Yaskawa INFORM job: BATMAN_2STR2.JBI

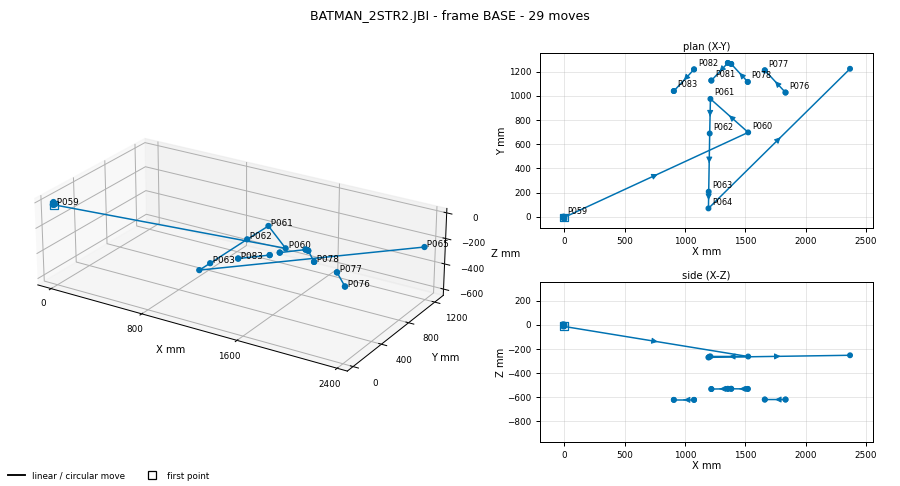
[picture p0: tool path of BATMAN_2STR2.JBI in frame BASE, 29 of 158 moves have a stored position in this frame; points joined in program order, loops and branches not executed]
/JOB
//NAME BATMAN_2STR2
///FOLDERNAME KRIS-SCIANA
//POS
///NPOS 87,87,0,38,0,0
///TOOL 0
///POSTYPE PULSE
///LIMIT ON
///PULSE
C00000=31537,-23080,-24186,7401,81948,158244
C00001=-4439,-79004,-57355,2552,77563,145804
C00002=-4909,-70479,-49283,2592,76991,145631
C00003=-4909,-70121,-48408,2595,76637,145623
C00004=-4003,-74801,-52630,2527,76803,145940
C00005=11747,-84119,-56660,1324,74120,151337
C00006=17222,-83520,-55007,884,73335,153227
C00007=17222,-83075,-54091,884,72998,153224
C00008=32420,-90805,-60082,-370,72663,158498
C00009=38310,-87672,-56905,-859,72363,160549
C00010=38411,-86269,-54218,-871,71436,160589
C00011=52965,-90491,-59465,-2036,72753,165631
C00012=61358,-83938,-55903,-2664,74169,168512
C00013=61358,-82452,-52843,-2677,73046,168534
C00014=75499,-77158,-53728,-3596,76905,173310
C00015=83067,-67878,-47888,-4094,78394,175877
C00016=83067,-67594,-47168,-4098,78099,175887
C00017=88580,-61652,-44685,-4402,79910,177718
C00018=88580,-61316,-43770,-4406,79520,177731
C00019=86164,-72702,-59256,-4234,83063,176784
C00020=57917,-53619,-44002,17021,94716,124656
C00021=59918,-45185,-32120,16966,91065,125425
C00022=59918,-44935,-31368,16961,90745,125381
C00023=57173,-65270,-44444,16695,89007,124177
C00024=59200,-80263,-49588,16922,84240,124236
C00025=59200,-79912,-48884,16927,83998,124202
C00026=59200,-86069,-61854,16879,88616,124838
C00027=77293,-89843,-63362,18058,83781,130525
C00028=78815,-87617,-60670,18129,82952,130941
C00029=78815,-87165,-59720,18140,82615,130890
C00030=77659,-102730,-69319,18171,80880,130220
C00031=85944,-117290,-70372,18932,72559,131861
C00032=85944,-116620,-69416,18956,72327,131824
C00033=85944,-124960,-81218,18696,75154,132276
C00034=151728,-153076,-87491,-11017,48359,191211
C00035=147386,-140874,-75268,-10077,46618,189610
C00036=147386,-140130,-74447,-10096,46496,189624
C00037=159688,-133609,-76919,-12343,52845,193892
C00038=159864,-112518,-69307,-11535,58898,193269
C00039=159864,-111881,-68341,-11567,58637,193296
C00040=178833,-115187,-73178,-14901,62898,200003
C00041=185982,-107062,-64617,-16080,63162,202660
C00042=185982,-103029,-58312,-16337,61422,202917
C00043=185982,-102236,-57075,-16389,61082,202968
C00044=187292,-93406,-58139,-15875,66332,202702
C00045=183818,-68327,-44618,-14942,70095,200919
C00046=183818,-67914,-43663,-14975,69731,200966
C00047=189068,-78650,-56857,-15464,73225,202429
C00048=240783,-65694,-51653,-5278,84394,164569
C00049=221621,-56342,-41396,-1214,76392,158122
C00050=221621,-56290,-41244,-1214,76326,158123
C00051=221621,-55882,-40078,-1216,75818,158128
C00052=209855,-65296,-47790,155,75648,154049
C00053=204224,-59057,-42452,814,75603,152098
C00054=204224,-58710,-41499,814,75195,152094
C00055=190935,-63343,-46423,2338,76108,147494
C00056=187139,-57536,-42749,2753,76951,146198
C00057=187139,-57216,-41822,2757,76545,146190
C00058=175859,-57355,-44220,3949,78417,142345
C00059=173058,-50767,-39052,4222,78764,141391
C00060=173058,-50451,-38053,4227,78312,141376
C00061=163443,-45354,-36848,5138,80747,138159
C00062=164371,-41258,-32523,5059,80134,138455
C00063=164371,-41027,-31730,5064,79765,138439
C00064=152450,-34091,-30773,6086,83554,134518
C00065=152482,-28025,-24496,6089,82810,134493
C00066=152482,-27812,-23636,6093,82393,134472
C00067=149914,-23676,-21598,6293,83456,133647
C00068=149914,-23406,-20465,6299,82902,133618
C00069=149914,-25053,-28729,6272,87116,133828
C00070=211398,-84605,-64904,-36,76260,154581
C00071=220860,-58623,-44430,-1132,77083,157849
C00072=149914,-25053,-28729,6272,87116,133828
C00073=120676,-124875,-96295,8199,80135,123403
C00074=-4439,-79004,-57355,2552,77563,145804
C00075=-4965,-72448,-51023,2596,77053,145613
C00076=88570,-66783,-53472,-4371,82677,177617
C00077=72474,-62045,-52325,1456,86059,123431
C00078=73182,-61072,-47349,1438,83485,123645
C00079=40588,-105091,-66546,14786,85577,117999
C00080=66697,-107157,-67194,17695,79826,126223
C00081=61032,-151860,-79989,18635,65463,124242
C00082=7538,-133985,-77466,26458,61671,147261
C00083=57429,-136223,-75586,15192,52650,153109
C00084=59881,-140929,-66526,16624,44527,152732
C00085=106253,-180552,-90268,3429,33706,171973
C00086=22771,-69913,-65485,-4348,88446,177417
///LIMIT OFF
BC00000=149550,282370,904111
BC00001=226428,281090,543192
BC00002=226428,281090,543192
BC00003=226428,281090,543192
BC00004=226427,281091,543189
BC00005=226427,281091,543189
BC00006=226427,281091,543189
BC00007=226427,281091,543189
BC00008=226427,281091,543189
BC00009=226427,281091,543189
BC00010=226427,281091,543189
BC00011=226427,281091,543189
BC00012=226427,281091,543189
BC00013=226427,281091,543189
BC00014=226427,281091,543189
BC00015=226427,281091,543189
BC00016=226427,281091,543189
BC00017=226427,281091,543189
BC00018=226427,281091,543189
BC00019=226427,281091,543187
BC00020=226427,281092,543184
BC00021=225242,280682,546364
BC00022=225242,280682,546364
BC00023=225242,280682,546364
BC00024=225242,280682,546364
BC00025=225242,280682,546364
BC00026=225242,280682,546364
BC00027=225242,280682,546364
BC00028=225242,280682,546364
BC00029=225242,280682,546364
BC00030=225242,280682,546364
BC00031=225242,280682,546364
BC00032=225242,280682,546364
BC00033=225242,280682,546364
BC00034=225242,280682,546364
BC00035=225242,280682,546364
BC00036=225242,280682,546364
BC00037=225242,280682,546364
BC00038=225242,280682,546364
BC00039=225242,280682,546364
BC00040=225242,280682,546364
BC00041=225242,280682,546364
BC00042=225242,280682,546364
BC00043=225242,280682,546364
BC00044=225242,280682,546364
BC00045=225242,280682,546364
BC00046=225242,280682,546364
BC00047=225242,280682,546364
BC00048=226427,281091,543187
BC00049=226427,319126,543187
BC00050=226427,319126,543187
BC00051=226427,319126,543187
BC00052=226427,319126,543184
BC00053=226427,319126,543184
BC00054=226427,319126,543184
BC00055=226427,319126,543184
BC00056=226427,319126,543184
BC00057=226427,319126,543184
BC00058=226427,319126,543184
BC00059=226427,319125,543182
BC00060=226427,319125,543182
BC00061=226427,319125,543182
BC00062=226427,319125,543182
BC00063=226427,319125,543182
BC00064=226427,319125,543182
BC00065=226427,319125,543182
BC00066=226427,319125,543182
BC00067=226427,319125,543182
BC00068=226427,319125,543182
BC00069=226427,319125,543182
BC00070=226427,319125,543182
BC00071=226427,319125,543182
BC00072=226427,319125,543182
BC00073=226427,319125,543182
BC00074=226428,281090,543192
BC00075=226428,281090,543192
BC00076=226428,281090,543192
BC00077=226428,281090,543192
BC00078=226428,281090,543192
BC00079=228873,257687,554679
BC00080=228873,257687,554679
BC00081=229563,251082,557921
BC00082=133596,251082,557921
BC00083=134171,249919,558492
BC00084=134171,249919,558492
BC00085=134170,249920,558489
BC00086=134714,456554,904710
///POSTYPE BASE
///RECTAN
///RCONF 0,0,0,0,0,0,0,0,0,0,0,0,0,0,0,0,0,0,0,0,0,0,0,0
P00059=-2.448,-6.714,-12.718,0.0000,0.0000,0.0000
P00060=1524.284,698.404,-261.973,-0.4635,36.8346,-1.2388
P00061=1211.499,975.999,-261.374,0.5148,35.2356,175.5099
P00062=1205.574,689.500,-262.704,0.5159,35.2461,175.5270
P00063=1197.217,207.358,-268.729,0.4863,35.2395,175.4586
P00064=1195.199,68.975,-269.171,0.5092,35.2366,175.4908
P00065=2367.684,1225.356,-251.745,0.6375,35.5356,-175.5535
P00070=2.449,-18.318,2.615,0.0000,0.0000,0.0000
P00071=-2.048,-0.034,-9.092,0.0000,0.0000,0.0000
P00072=-1.595,-0.049,-6.373,0.0000,0.0000,0.0000
P00073=-8.474,-10.331,-11.894,0.0000,0.0000,0.0000
P00074=1.731,-3.007,-10.460,0.0000,0.0000,0.0000
///RCONF 0,1,0,0,0,0,0,0,0,0,0,0,0,0,0,0,0,0,0,0,0,0,0,0
P00075=-9.634,0.014,4.922,0.0000,0.0000,0.0000
///RCONF 0,0,0,0,0,0,0,0,0,0,0,0,0,0,0,0,0,0,0,0,0,0,0,0
P00076=1833.500,1028.615,-618.215,10.0256,37.5190,56.2681
P00077=1661.766,1212.555,-618.325,10.0309,37.5577,56.2858
P00078=1520.740,1116.757,-530.271,10.0398,37.5578,56.2925
P00079=1383.754,1265.334,-529.217,10.0293,37.5461,56.2787
P00080=1355.833,1273.708,-529.583,10.0283,37.5305,126.4716
P00081=1219.184,1127.874,-531.327,10.0137,37.5345,126.4324
P00082=1075.995,1220.294,-620.895,10.0203,37.5289,126.4576
P00083=908.434,1040.970,-620.895,10.0141,37.5419,126.4584
P00087=-17.000,-22.000,-3.000,0.0000,0.0000,0.0000
P00088=-8.588,-0.108,-11.097,0.0000,0.0000,0.0000
P00089=5.931,-12.286,-8.772,0.0000,0.0000,0.0000
P00090=-14.057,13.261,-6.464,0.0000,0.0000,0.0000
P00091=1.048,0.648,3.624,0.0000,0.0000,0.0000
P00092=12.000,-9.000,-4.000,0.0000,0.0000,0.0000
P00093=-12.000,12.000,-3.000,0.0000,0.0000,0.0000
P00094=10.000,10.000,-3.000,0.0000,0.0000,0.0000
P00095=-11.943,-14.820,-6.815,0.0000,0.0000,0.0000
P00096=-4.844,-19.262,-10.890,0.0000,0.0000,0.0000
P00108=0.000,0.000,-3.000,0.0000,0.0000,0.0000
P00123=0.000,-50.000,0.000,0.0000,0.0000,0.0000
P00125=0.000,0.000,2.400,0.0000,0.0000,0.0000
P00126=-50.000,0.000,0.000,0.0000,0.0000,0.0000
P00127=50.000,0.000,0.000,0.0000,0.0000,0.0000
P00172=2.000,-12.000,-3.000,0.0000,0.0000,40.0000
P00173=-5.000,-9.000,-2.400,0.0000,0.0000,-15.0000
//INST
///DATE 2024/07/30 17:34
///COMM NOWY SEARCH
///ATTR SC,RW
///GROUP1 RB1,BS1
NOP
SFTOF
MOVJ C00000 BC00000 VJ=60.00
MOVJ C00001 BC00001 VJ=60.00
'POMIAR PRAWA STRONA
'1
MOVL C00002 BC00002 V=166.7
MOVL C00003 BC00003 V=16.7 PL=0 SRCH RIN#(1)=ON T=1.00 DIS=20.0
TIMER T=0.20
IMOV P125 V=13.3 PL=0
TIMER T=0.20
IMOV P127 V=13.3 PL=0 SRCH RIN#(1)=ON DIS=20.0
TIMER T=0.20
GETS PX070 $PX001
TIMER T=0.10
MOVJ C00004 BC00004 VJ=15.00
MOVJ C00005 BC00005 VJ=15.00
'2
MOVL C00006 BC00006 V=50.0
MOVL C00007 BC00007 V=16.7 PL=0 SRCH RIN#(1)=ON T=1.00 DIS=20.0
TIMER T=0.20
IMOV P125 V=13.3 PL=0
TIMER T=0.20
IMOV P127 V=13.3 PL=0 SRCH RIN#(1)=ON DIS=20.0
TIMER T=0.20
GETS PX071 $PX001
TIMER T=0.10
MOVJ C00008 BC00008 VJ=15.00
'3
MOVL C00009 BC00009 V=50.0
MOVL C00010 BC00010 V=16.7 PL=0 SRCH RIN#(1)=ON T=1.00 DIS=20.0
TIMER T=0.20
IMOV P125 V=13.3 PL=0
TIMER T=0.20
IMOV P127 V=13.3 PL=0 SRCH RIN#(1)=ON DIS=20.0
TIMER T=0.20
GETS PX072 $PX001
TIMER T=0.10
MOVJ C00011 BC00011 VJ=15.00
'4
MOVL C00012 BC00012 V=50.0
MOVL C00013 BC00013 V=16.7 PL=0 SRCH RIN#(1)=ON T=1.00 DIS=20.0
TIMER T=0.20
IMOV P125 V=13.3 PL=0
TIMER T=0.20
IMOV P127 V=13.3 PL=0 SRCH RIN#(1)=ON DIS=20.0
TIMER T=0.20
GETS PX073 $PX001
TIMER T=0.10
MOVJ C00014 BC00014 VJ=15.00
'5
MOVL C00015 BC00015 V=50.0
MOVL C00016 BC00016 V=16.7 PL=0 SRCH RIN#(1)=ON T=1.00 DIS=20.0
TIMER T=0.20
IMOV P125 V=13.3 PL=0
TIMER T=0.20
IMOV P127 V=13.3 PL=0 SRCH RIN#(1)=ON DIS=20.0
TIMER T=0.20
GETS PX074 $PX001
TIMER T=0.10
MOVL C00017 BC00017 V=50.0
MOVL C00018 BC00018 V=16.7 PL=0 SRCH RIN#(1)=ON T=1.00 DIS=20.0
TIMER T=0.20
IMOV P125 V=13.3 PL=0
TIMER T=0.20
IMOV P127 V=13.3 PL=0 SRCH RIN#(1)=ON DIS=20.0
TIMER T=0.20
GETS PX075 $PX001
TIMER T=0.10
MOVJ C00019 BC00019 VJ=15.00
MOVJ C00020 BC00020 VJ=30.00
'POMIAR BATMAN
MOVL C00021 BC00021 V=166.7
MOVL C00022 BC00022 V=16.7 PL=0 SRCH RIN#(1)=ON T=1.00 DIS=20.0
TIMER T=0.20
IMOV P125 V=13.3 PL=0
TIMER T=0.20
IMOV P123 V=13.3 PL=0 SRCH RIN#(1)=ON DIS=20.0
TIMER T=0.20
GETS PX076 $PX001
TIMER T=0.10
MOVJ C00023 BC00023 VJ=30.00
MOVL C00024 BC00024 V=166.7
MOVL C00025 BC00025 V=16.7 PL=0 SRCH RIN#(1)=ON T=1.00 DIS=20.0
TIMER T=0.20
IMOV P125 V=13.3 PL=0
TIMER T=0.20
IMOV P123 V=13.3 PL=0 SRCH RIN#(1)=ON DIS=20.0
TIMER T=0.20
GETS PX077 $PX001
TIMER T=0.10
MOVJ C00026 BC00026 VJ=30.00
MOVJ C00027 BC00027 VJ=30.00
MOVL C00028 BC00028 V=166.7
MOVL C00029 BC00029 V=16.7 PL=0 SRCH RIN#(1)=ON T=1.00 DIS=20.0
TIMER T=0.20
IMOV P125 V=13.3 PL=0
TIMER T=0.20
IMOV P123 V=13.3 PL=0 SRCH RIN#(1)=ON DIS=20.0
TIMER T=0.20
GETS PX078 $PX001
TIMER T=0.10
MOVJ C00030 BC00030 VJ=30.00
MOVL C00031 BC00031 V=166.7
MOVL C00032 BC00032 V=16.7 PL=0 SRCH RIN#(1)=ON T=1.00 DIS=20.0
TIMER T=0.20
IMOV P125 V=13.3 PL=0
TIMER T=0.20
IMOV P123 V=13.3 PL=0 SRCH RIN#(1)=ON DIS=20.0
TIMER T=0.20
GETS PX079 $PX001
TIMER T=0.10
MOVJ C00033 BC00033 VJ=30.00
MOVJ C00034 BC00034 VJ=30.00
MOVL C00035 BC00035 V=166.7
MOVL C00036 BC00036 V=16.7 PL=0 SRCH RIN#(1)=ON T=1.00 DIS=20.0
TIMER T=0.20
IMOV P125 V=13.3 PL=0
TIMER T=0.20
IMOV P123 V=13.3 PL=0 SRCH RIN#(1)=ON DIS=20.0
TIMER T=0.20
GETS PX080 $PX001
TIMER T=0.10
MOVJ C00037 BC00037 VJ=30.00
MOVL C00038 BC00038 V=166.7
MOVL C00039 BC00039 V=16.7 PL=0 SRCH RIN#(1)=ON T=1.00 DIS=20.0
TIMER T=0.20
IMOV P125 V=13.3 PL=0
TIMER T=0.20
IMOV P123 V=13.3 PL=0 SRCH RIN#(1)=ON DIS=20.0
TIMER T=0.20
GETS PX081 $PX001
TIMER T=0.10
MOVJ C00040 BC00040 VJ=30.00
MOVJ C00041 BC00041 VJ=30.00
MOVL C00042 BC00042 V=166.7
MOVL C00043 BC00043 V=16.7 PL=0 SRCH RIN#(1)=ON T=1.00 DIS=20.0
TIMER T=0.20
IMOV P125 V=13.3 PL=0
TIMER T=0.20
IMOV P123 V=13.3 PL=0 SRCH RIN#(1)=ON DIS=20.0
TIMER T=0.20
GETS PX082 $PX001
TIMER T=0.10
MOVJ C00044 BC00044 VJ=30.00
MOVL C00045 BC00045 V=166.7
MOVL C00046 BC00046 V=16.7 PL=0 SRCH RIN#(1)=ON T=1.00 DIS=20.0
TIMER T=0.20
IMOV P125 V=13.3 PL=0
TIMER T=0.20
IMOV P123 V=13.3 PL=0 SRCH RIN#(1)=ON DIS=20.0
TIMER T=0.20
GETS PX083 $PX001
TIMER T=0.10
MOVJ C00047 BC00047 VJ=30.00
'KONIEC POMIAR BATMAN 1STR
SFTOF
MOVJ C00048 BC00048 VJ=50.00
SFTOF
MOVJ C00049 BC00049 VJ=15.00
'1
MOVL C00050 BC00050 V=166.7
MOVL C00051 BC00051 V=16.7 PL=0 SRCH RIN#(1)=ON T=1.00 DIS=20.0
TIMER T=0.20
IMOV P125 V=13.3 PL=0
TIMER T=0.20
IMOV P126 V=13.3 PL=0 SRCH RIN#(1)=ON DIS=20.0
TIMER T=0.20
GETS PX059 $PX001
TIMER T=0.10
MOVJ C00052 BC00052 VJ=15.00
MOVL C00053 BC00053 V=166.7
MOVL C00054 BC00054 V=16.7 PL=0 SRCH RIN#(1)=ON T=1.00 DIS=20.0
TIMER T=0.20
IMOV P125 V=13.3 PL=0
TIMER T=0.20
IMOV P126 V=13.3 PL=0 SRCH RIN#(1)=ON DIS=20.0
TIMER T=0.20
GETS PX060 $PX001
TIMER T=0.10
MOVJ C00055 BC00055 VJ=50.00
'2
MOVL C00056 BC00056 V=50.0
MOVL C00057 BC00057 V=16.7 PL=0 SRCH RIN#(1)=ON T=1.00 DIS=30.0
TIMER T=0.20
IMOV P125 V=13.3 PL=0
TIMER T=0.20
IMOV P126 V=13.3 PL=0 SRCH RIN#(1)=ON DIS=20.0
TIMER T=0.20
GETS PX061 $PX001
TIMER T=0.10
MOVJ C00058 BC00058 VJ=50.00
'3
MOVL C00059 BC00059 V=50.0
MOVL C00060 BC00060 V=16.7 PL=0 SRCH RIN#(1)=ON T=1.00 DIS=30.0
TIMER T=0.20
IMOV P125 V=13.3 PL=0
TIMER T=0.20
IMOV P126 V=13.3 PL=0 SRCH RIN#(1)=ON DIS=20.0
TIMER T=0.20
GETS PX062 $PX001
TIMER T=0.10
MOVJ C00061 BC00061 VJ=50.00
'4
MOVL C00062 BC00062 V=50.0
MOVL C00063 BC00063 V=16.7 PL=0 SRCH RIN#(1)=ON T=1.00 DIS=30.0
TIMER T=0.20
IMOV P125 V=13.3 PL=0
TIMER T=0.20
IMOV P126 V=13.3 PL=0 SRCH RIN#(1)=ON DIS=20.0
TIMER T=0.20
GETS PX063 $PX001
TIMER T=0.10
MOVJ C00064 BC00064 VJ=15.00
'5
MOVL C00065 BC00065 V=50.0
MOVL C00066 BC00066 V=16.7 PL=0 SRCH RIN#(1)=ON T=1.00 DIS=20.0
TIMER T=0.20
IMOV P125 V=13.3 PL=0
TIMER T=0.20
IMOV P126 V=13.3 PL=0 SRCH RIN#(1)=ON DIS=20.0
TIMER T=0.20
GETS PX064 $PX001
TIMER T=0.10
MOVL C00067 BC00067 V=50.0
MOVL C00068 BC00068 V=16.7 PL=0 SRCH RIN#(1)=ON T=1.00 DIS=20.0
TIMER T=0.20
IMOV P125 V=13.3 PL=0
TIMER T=0.20
IMOV P126 V=13.3 PL=0 SRCH RIN#(1)=ON DIS=20.0
TIMER T=0.20
GETS PX065 $PX001
TIMER T=0.10
MOVJ C00069 BC00069 VJ=15.00
'********
'********
'********
MOVJ C00070 BC00070 VJ=15.00
MOVL C00071 BC00071 V=333.3
MACRO1 MJ#(0) ARGF7
SFTOF
SFTON P095
MOVL P059 V=83.3
ARCON
MOVL P060 V=10.8
MOVL P061 V=10.8
ARCON
MOVL P062 V=10.8
MOVL P063 V=10.8
MOVL P064 V=10.8
SFTOF
SFTON P172
MOVL P065 V=10.8
ARCOF
MOVJ C00072 BC00072 VJ=15.00
SFTOF
MOVJ C00073 BC00073 VJ=15.00
MOVJ C00074 BC00074 VJ=40.00
SFTON P096
MOVJ C00075 BC00075 VJ=15.00
MOVL P070 V=83.3
ARCON
MOVL P071 V=10.8
MOVL P072 V=10.8
MOVL P073 V=10.8
MOVL P074 V=10.8
SFTOF
SFTON P173
MOVL P075 V=10.8
ARCOF
SFTOF
MOVJ C00076 BC00076 VJ=15.00
MOVJ C00077 BC00077 VJ=30.00
'START SPAWANIE BATMAN
MOVJ C00078 BC00078 VJ=30.00
SFTON P090
MOVL P076 V=83.3
SFTOF
ARCON
SFTON P108
ARCON
MOVL P076 V=10.8
MOVL P077 V=10.8
SFTOF
SFTON P091
MOVL P077 V=10.8
ARCOF
SFTOF
MOVJ C00079 BC00079 VJ=30.00
MOVJ C00080 BC00080 VJ=30.00
SFTON P092
MOVL P078 V=83.3
ARCON
SFTOF
SFTON P108
MOVL P078 V=10.8
MOVL P079 V=10.8
SFTOF
SFTON P093
MOVL P079 V=10.8
ARCOF
SFTOF
MOVJ C00081 BC00081 VJ=30.00
MOVJ C00082 BC00082 VJ=30.00
SFTON P094
MOVL P080 V=83.3
SFTOF
ARCON
SFTON P108
MOVL P080 V=10.8
MOVL P081 V=10.8
SFTOF
SFTON P087
MOVL P081 V=10.8
SFTOF
ARCOF
MOVJ C00083 BC00083 VJ=30.00
MOVJ C00084 BC00084 VJ=30.00
SFTON P088
MOVL P082 V=83.3
SFTOF
ARCON
SFTON P108
MOVL P082 V=10.8
MOVL P083 V=10.8
SFTOF
SFTON P089
MOVL P083 V=10.8
SFTOF
ARCOF
MOVJ C00085 BC00085 VJ=30.00
MOVJ C00086 BC00086 VJ=100.00
CALL JOB:ONLYCUT-R1_LONG
END
